% RSLogix 500 project UNTITLED.RSS, saved by version 8.40.00.08 %
PROJECT "UNTITLED"    % processor: MicroLogix 1000 %

PROGRAM FILES
  LAD 2 "MAIN_PROG"  6 rungs
  LAD 3 "USER_FAULT"  1 rungs
  LAD 4 "HSC_INT"  1 rungs
  LAD 5 "STI_INT"  1 rungs
  LAD 6, 7, 8, 9, 10, 11, 12, 13, 14, 15, 16: only END

DATA FILES
  O0 OUTPUT  1 elements
  I1 INPUT  2 elements
  S2 STATUS  33 elements
  B3 BINARY  32 elements
  T4 TIMER  40 elements
  C5 COUNTER  32 elements
  R6 CONTROL  16 elements
  N7 INTEGER  105 elements

LADDER 2 "MAIN_PROG"
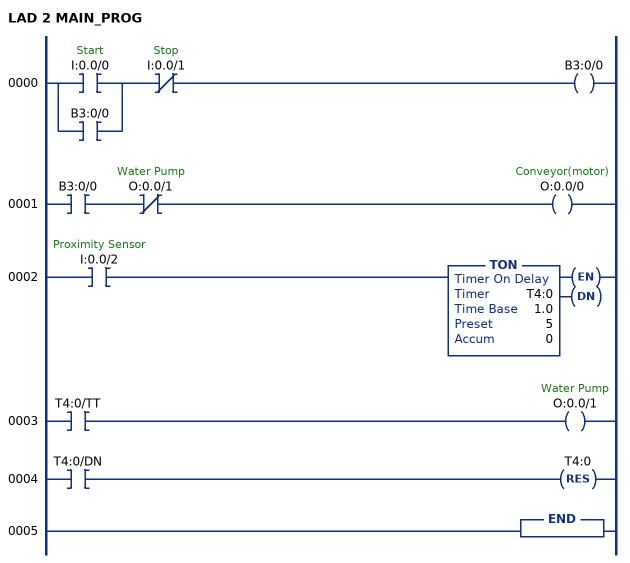
% Rung: 0 %
SOR BST XIC I:0.0/0 NXB XIC B3:0/0 BND XIO I:0.0/1 OTE B3:0/0 EOR
%   I:0.0/0  "Start" %
%   I:0.0/1  "Stop" %
% Rung: 1 %
SOR XIC B3:0/0 XIO O:0.0/1 OTE O:0.0/0 EOR
%   O:0.0/1  "Water Pump" %
%   O:0.0/0  "Conveyor(motor)" %
% Rung: 2 %
SOR XIC I:0.0/2 TON T4:0 1.0 5 0 EOR
%   I:0.0/2  "Proximity Sensor" %
% Rung: 3 %
SOR XIC T4:0/TT OTE O:0.0/1 EOR
%   O:0.0/1  "Water Pump" %
% Rung: 4 %
SOR XIC T4:0/DN RES T4:0 EOR
% Rung: 5 %
SOR END EOR

DATA TABLE (non-zero values as saved)
DATA T4
% .PRE .ACC %
% T4:0 % 5 0
